// TIA Portal V16 export
// export: Created 2024-05-13T12:49:09.5234335Z, ExportSetting WithDefaults, DisplayName Totally Integrated Automation Portal, DisplayVersion V16 Update 6, DisplayName TIA Portal Version Control Interface, DisplayVersion V16 Update 2, DisplayName TIA Portal Openness, DisplayVersion V16 Update 6, DisplayName TIA Portal Test Suite Advanced, DisplayVersion V16, DisplayName SINAMICS Startdrive Advanced, DisplayVersion V16 Update 5, DisplayName SINAMICS Startdrive G130, G150, S120, S150, SINAMICS MV, S210, DisplayVersion V16 Update 5, DisplayName SINAMICS Startdrive G110M, G120, G120C, G120D, G120P, G115D, DisplayVersion V16 Update 5, DisplayName STEP 7 Professional, DisplayVersion V16 Update 6, DisplayName STEP 7 Safety, DisplayVersion V16, DisplayName WinCC Advanced, DisplayVersion V16 Update 6
TYPE "SCA_rotatingRollers_flags"
// stored: IsFailsafeCompliant false
   STRUCT
      Speed_1 : Bool;   // Speed selection 1
      Speed_2 : Bool;   // Speed selection 2
      Speed_3 : Bool;   // Speed selection 3
      Speed_4 : Bool;   // Speed selection 4
      Marking_Done : Bool;   // Belly Marking Done
      Marking_Trigger : Bool;   // Print head Trigger
      Device_stopped : Bool;
   END_STRUCT;
END_TYPE
